FUNCTION_BLOCK FB_TimeStampBuffer
(*
    A Companion to FB_LREALBuffer that accumulates timestamps
    2019-10-09 Zachary Lentz
*)
VAR_INPUT
    // If TRUE, we'll accumulate a value on this cycle.
    bExecute: BOOL;
END_VAR
VAR_OUTPUT
    afOutput: ARRAY [1..1000] OF LREAL;
    bNewArray: BOOL;
END_VAR
VAR
    fbUnixTime: FB_UnixTimestamp;
    fbLREALBuffer: FB_LREALBuffer;
END_VAR

fbUnixTime(
    bExecute := bExecute,
    fTime => fbLREALBuffer.fInput);
fbLREALBuffer(
    bExecute := bExecute,
    afOutput => afOutput,
    bNewArray => bNewArray);

END_FUNCTION_BLOCK

(* stored: Version 1.1.0.1
   POU FB_TimeStampBuffer: Id {b2db97ec-7312-4822-a3b4-76ec1968b59f}, SpecialFunc None *)
